SUBAPPLICATION Baumzaehler (* Baumzaehler: zaehlt die gepflanzten Baeume hoch/runter, speichert den Zaehlerstand persistent im NVS und zeigt ihn auf dem Terminal an *)
  (* Standard: 61499-2 *)
  (* Version 1.0, 2024-10-09, Elias *)
  PACKAGE FBs::Baumsetzer::func::Zaehlermenue;
  IMPORT NVS_Keys::Key_Baumzaehler_Store;
  IMPORT test::FBs::Baumsetzer::Constants::DefaultPool;
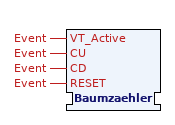
  EVENT_INPUT
    VT_Active; (* Terminal aktiv (Aktualisierung der Anzeige anfordern) *)
    CU; (* Counts up *)
    CD; (* Zaehlerstand herunterzaehlen *)
    RESET; (* Resets Value *)
  END_EVENT
  SUBAPPS
    Baumzaehler : Zaehler(KEY := Key_Baumzaehler_Store, u16ObjId := DefaultPool::NumberVariable_Baumzaehler);
  END_SUBAPPS
  EVENT_CONNECTIONS
    RESET TO Baumzaehler.R;
    CU TO Baumzaehler.CU;
    CD TO Baumzaehler.CD;
    VT_Active TO Baumzaehler.rVT;
  END_CONNECTIONS
END_SUBAPPLICATION
